// LS Electric XG5000 project: 25.센서 활용 자재 구별 제어
// PLC NewPLC
// module base 0 slot 0: 입출력 모듈:XBM-DN/DP32HP (DC 24V입력/TR 출력, 32점)
// module base 0 slot 2: 입력 모듈:XBE-DC08A (DC 24V 입력, 8점 (전류소스 싱크공용))

PROGRAM NewProgram (task: 스캔 프로그램)

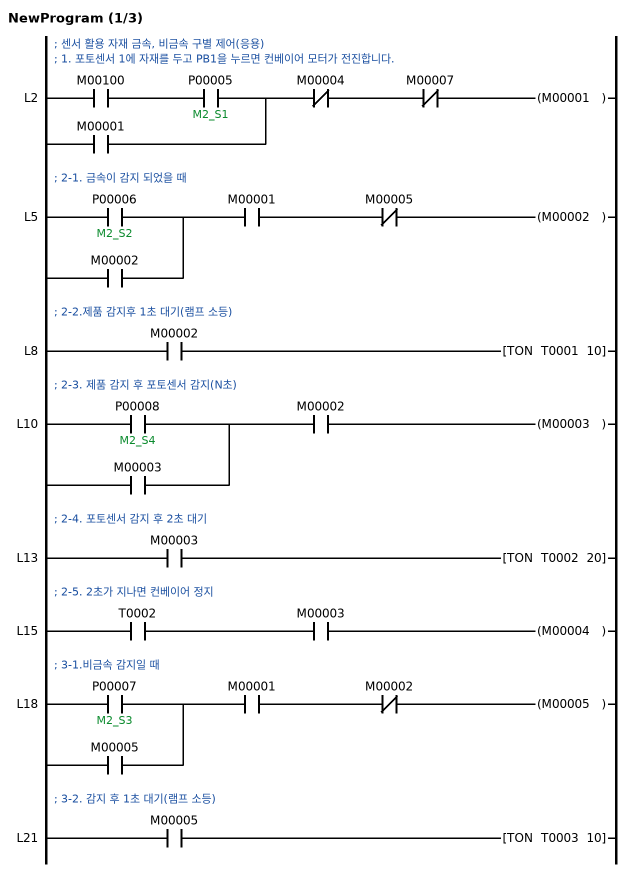
// 센서 활용 자재 금속, 비금속 구별 제어(응용)
// 1. 포토센서 1에 자재를 두고 PB1을 누르면 컨베이어 모터가 전진합니다.
; L2
LOAD      M00100
AND       P00005	// M2_S1
OR        M00001
AND NOT   M00004
AND NOT   M00007
OUT       M00001
// 2-1. 금속이 감지 되었을 때
; L5
LOAD      P00006	// M2_S2
OR        M00002
AND       M00001
AND NOT   M00005
OUT       M00002
// 2-2.제품 감지후 1초 대기(램프 소등)
; L8
LOAD      M00002
TON       T0001 10
// 2-3. 제품 감지 후 포토센서 감지(N초)
; L10
LOAD      P00008	// M2_S4
OR        M00003
AND       M00002
OUT       M00003
// 2-4. 포토센서 감지 후 2초 대기
; L13
LOAD      M00003
TON       T0002 20
// 2-5. 2초가 지나면 컨베이어 정지
; L15
LOAD      T0002
AND       M00003
OUT       M00004
// 3-1.비금속 감지일 때
; L18
LOAD      P00007	// M2_S3
OR        M00005
AND       M00001
AND NOT   M00002
OUT       M00005
// 3-2. 감지 후 1초 대기(램프 소등)
; L21
LOAD      M00005
TON       T0003 10

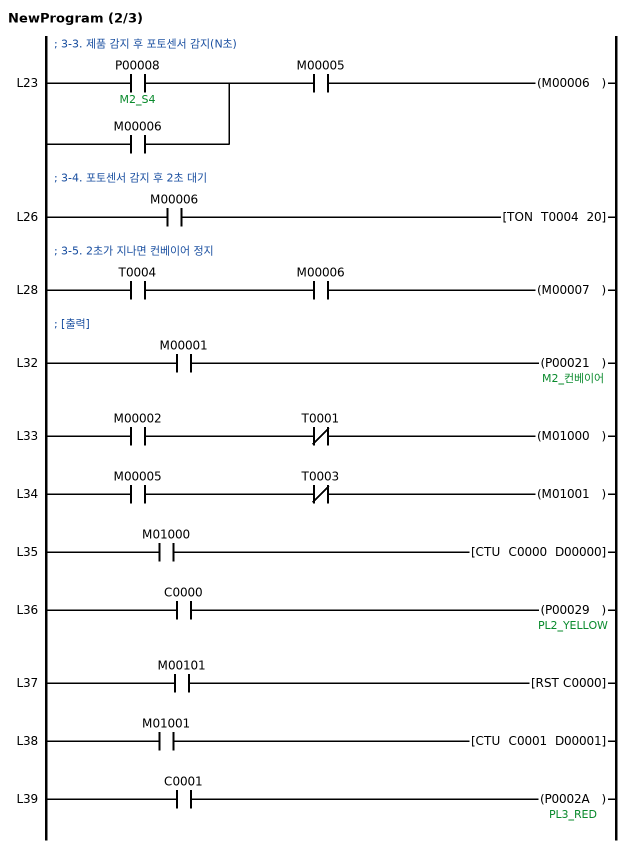
// 3-3. 제품 감지 후 포토센서 감지(N초)
; L23
LOAD      P00008	// M2_S4
OR        M00006
AND       M00005
OUT       M00006
// 3-4. 포토센서 감지 후 2초 대기
; L26
LOAD      M00006
TON       T0004 20
// 3-5. 2초가 지나면 컨베이어 정지
; L28
LOAD      T0004
AND       M00006
OUT       M00007
// [출력]
; L32
LOAD      M00001
OUT       P00021	// M2_컨베이어
; L33
LOAD      M00002
AND NOT   T0001
OUT       M01000
; L34
LOAD      M00005
AND NOT   T0003
OUT       M01001
; L35
LOAD      M01000
CTU       C0000 D00000
; L36
LOAD      C0000
OUT       P00029	// PL2_YELLOW
; L37
LOAD      M00101
RST       C0000
; L38
LOAD      M01001
CTU       C0001 D00001
; L39
LOAD      C0001
OUT       P0002A	// PL3_RED

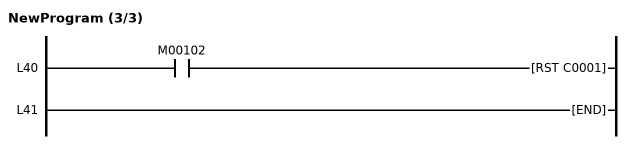
; L40
LOAD      M00102
RST       C0001
; L41
END

VARIABLES AND COMMENTS (devices not used above)
P00080	BIT	PB1
P00081	BIT	PB2
P00028	BIT	PL1_GREEN
P00083	BIT	PB4
P00082	BIT	PB3
P00020	BIT	M1_SOL1
P00000	BIT	M1_CS1
P00001	BIT	M1_CS2
P00002	BIT	M1_S1
P00003	BIT	M2_CS1
P00023	BIT	M2_SOL1
P00004	BIT	M2_CS2
P00024	BIT	M2_가공모터